// TIA Portal V18 export
FUNCTION "AHUSustainedSummaryRequests" : Void   // FC60103, LAD
{ S7_Optimized_Access := 'TRUE' }
VERSION : 0.1
// stored: AutoNumber false, IsIECCheckEnabled false, SetENOAutomatically false, UDAEnableTagReadback false
   VAR_INPUT
      iUnitID : Int;
      xNightCoolingRequest : Bool;
      xSustainedOnCoolingRequest : Bool;
      xSustainedOnHeatingRequest : Bool;
      xSustainedOnIAQRequest : Bool;
      xSustainedOnBuildingdPRequest : Bool;
      xAlarmFrostBlocking : Bool;
      xAlarmBlocking : Bool;
   END_VAR
   VAR_OUTPUT
      cSummaryTempRequest : Byte;
      xStartRequest : Bool;
      xBlockRequest : Bool;
   END_VAR
BEGIN

REGION Network 1 (SCL)
   #xStartRequest := #xNightCoolingRequest OR
   #xSustainedOnCoolingRequest OR
   #xSustainedOnHeatingRequest OR  
   #xSustainedOnIAQRequest OR
   #xSustainedOnBuildingdPRequest;
END_REGION

REGION Network 2 (SCL)
   #xBlockRequest := #xAlarmFrostBlocking OR
   #xAlarmBlocking;
END_REGION

REGION Network 3 (SCL)
   IF #xNightCoolingRequest THEN
       #cSummaryTempRequest := 3;
   ELSIF #xSustainedOnCoolingRequest THEN
       #cSummaryTempRequest := 2;
   ELSE
       IF #xSustainedOnHeatingRequest THEN
           #cSummaryTempRequest := 1;
       ELSE
           #cSummaryTempRequest := 0;
       END_IF;

   END_IF;
END_REGION
END_FUNCTION
